// TIA Portal V17 export
// export: Created 2022-07-20T07:02:42.7612496Z, ExportSetting WithDefaults, DisplayName Totally Integrated Automation Portal, DisplayVersion V17, DisplayName TIA Portal Openness, DisplayVersion V17, DisplayName TIA Portal Version Control Interface, DisplayVersion V17, DisplayName SINAMICS Startdrive Advanced, DisplayVersion V17, DisplayName SINAMICS Startdrive G130, G150, S120, S150, SINAMICS MV, S210, DisplayVersion V17, DisplayName SINAMICS Startdrive G110M, G120, G120C, G120D, G120P, G115D, DisplayVersion V17, DisplayName STEP 7 Professional, DisplayVersion V17, DisplayName STEP 7 Safety, DisplayVersion V17, DisplayName WinCC Advanced, DisplayVersion V17
DATA_BLOCK "DataExample1"   // DB1
{ S7_Optimized_Access := 'TRUE' }
VERSION : 0.1
// stored: AutoNumber true, DBAccessibleFromOPCUA true, IsOnlyStoredInLoadMemory false, IsRetainMemResEnabled false, IsWriteProtectedInAS false, MemoryReserve 100
   VAR
      hscData { S7_SetPoint := 'True'} : HSC_Period;   // Instruction CTRL_HSC_EXT: CTRL
      hscDone : Bool;   // Instruction CTRL_HSC_EXT: Done
      hscBusy : Bool;   // Instruction CTRL_HSC_EXT: Busy
      hscError : Bool;   // Instruction CTRL_HSC_EXT: Error
      hscStatus : Word;   // Instruction CTRL_HSC_EXT: Status
      numPulsePerRot : Int := 1000;   // Number of pulses per rotation
      overflow : Bool;   // Elapsed time overflow
      speed : Real := 0.0;   // Calculated speed [rpm]
      vitesse : Real;
   END_VAR
BEGIN
   hscData.EnHSC := TRUE;
   hscData.NewPeriod := 10;
END_DATA_BLOCK
